// TIA Portal V19 export
FUNCTION "SUGAR" : Void   // FC21, LAD
{ S7_Optimized_Access := 'TRUE' }
// stored: SetENOAutomatically false
   VAR_TEMP   // added for the SCL form of the ladder/FBD networks
      _w1 : Bool;
   END_VAR
BEGIN

REGION Network 1: START MFG PROCESS //////////////////////////////
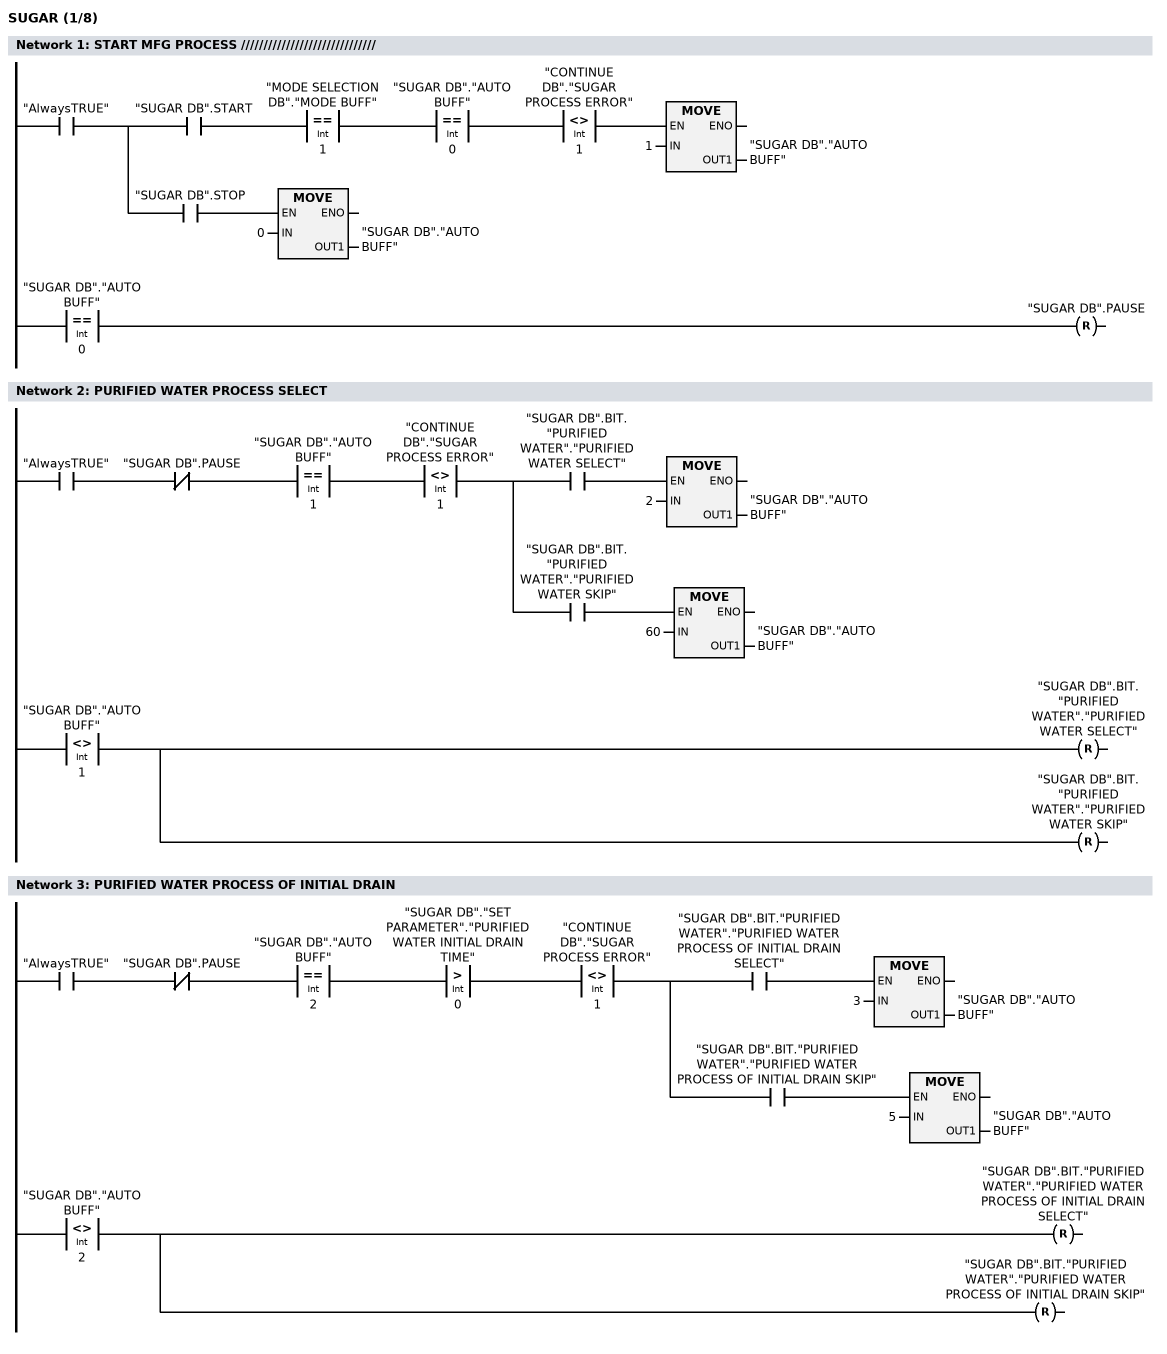
   RUNG wire#powerrail
      Contact( "AlwaysTRUE" )
      wire#w1
      Contact( "SUGAR DB".START )
      { S7_Templates := "SrcType := Int" } EQ_Contact(in1 := "MODE SELECTION DB"."MODE BUFF", in2 := 1)
      { S7_Templates := "SrcType := Int" } EQ_Contact(in1 := "SUGAR DB"."AUTO BUFF", in2 := 0)
      { S7_Templates := "SrcType := Int" } NE_Contact(in1 := "CONTINUE DB"."SUGAR PROCESS ERROR", in2 := 1)
      Move(in := 1, out1 => "SUGAR DB"."AUTO BUFF")
   END_RUNG
   RUNG wire#w1
      Contact( "SUGAR DB".STOP )
      Move(in := 0, out1 => "SUGAR DB"."AUTO BUFF")
   END_RUNG
   RUNG wire#powerrail
      { S7_Templates := "SrcType := Int" } EQ_Contact(in1 := "SUGAR DB"."AUTO BUFF", in2 := 0)
      R_Coil( "SUGAR DB".PAUSE )
   END_RUNG
   // the same network as SCL:
   IF "AlwaysTRUE" AND "SUGAR DB".START AND ("MODE SELECTION DB"."MODE BUFF" = 1) AND ("SUGAR DB"."AUTO BUFF" = 0) AND ("CONTINUE DB"."SUGAR PROCESS ERROR" <> 1) THEN
       "SUGAR DB"."AUTO BUFF" := 1;
   END_IF;
   IF "AlwaysTRUE" AND "SUGAR DB".STOP THEN "SUGAR DB"."AUTO BUFF" := 0; END_IF;
   IF "SUGAR DB"."AUTO BUFF" = 0 THEN "SUGAR DB".PAUSE := FALSE; END_IF;
END_REGION

REGION Network 2: PURIFIED WATER PROCESS SELECT
   RUNG wire#powerrail
      Contact( "AlwaysTRUE" )
      I_Contact( "SUGAR DB".PAUSE )
      { S7_Templates := "SrcType := Int" } EQ_Contact(in1 := "SUGAR DB"."AUTO BUFF", in2 := 1)
      { S7_Templates := "SrcType := Int" } NE_Contact(in1 := "CONTINUE DB"."SUGAR PROCESS ERROR", in2 := 1)
      wire#w1
      Contact( "SUGAR DB".BIT."PURIFIED WATER"."PURIFIED WATER SELECT" )
      Move(in := 2, out1 => "SUGAR DB"."AUTO BUFF")
   END_RUNG
   RUNG wire#w1
      Contact( "SUGAR DB".BIT."PURIFIED WATER"."PURIFIED WATER SKIP" )
      Move(in := 60, out1 => "SUGAR DB"."AUTO BUFF")
   END_RUNG
   RUNG wire#powerrail
      { S7_Templates := "SrcType := Int" } NE_Contact(in1 := "SUGAR DB"."AUTO BUFF", in2 := 1)
      wire#w2
      R_Coil( "SUGAR DB".BIT."PURIFIED WATER"."PURIFIED WATER SELECT" )
   END_RUNG
   RUNG wire#w2
      R_Coil( "SUGAR DB".BIT."PURIFIED WATER"."PURIFIED WATER SKIP" )
   END_RUNG
   // the same network as SCL:
   #_w1 := "AlwaysTRUE" AND NOT "SUGAR DB".PAUSE AND ("SUGAR DB"."AUTO BUFF" = 1) AND ("CONTINUE DB"."SUGAR PROCESS ERROR" <> 1);
   IF #_w1 AND "SUGAR DB".BIT."PURIFIED WATER"."PURIFIED WATER SELECT" THEN
       "SUGAR DB"."AUTO BUFF" := 2;
   END_IF;
   IF #_w1 AND "SUGAR DB".BIT."PURIFIED WATER"."PURIFIED WATER SKIP" THEN
       "SUGAR DB"."AUTO BUFF" := 60;
   END_IF;
   IF "SUGAR DB"."AUTO BUFF" <> 1 THEN
       "SUGAR DB".BIT."PURIFIED WATER"."PURIFIED WATER SELECT" := FALSE;
       "SUGAR DB".BIT."PURIFIED WATER"."PURIFIED WATER SKIP" := FALSE;
   END_IF;
END_REGION

REGION Network 3: PURIFIED WATER PROCESS OF INITIAL DRAIN
   RUNG wire#powerrail
      Contact( "AlwaysTRUE" )
      I_Contact( "SUGAR DB".PAUSE )
      { S7_Templates := "SrcType := Int" } EQ_Contact(in1 := "SUGAR DB"."AUTO BUFF", in2 := 2)
      { S7_Templates := "SrcType := Int" } GT_Contact(in1 := "SUGAR DB"."SET PARAMETER"."PURIFIED WATER INITIAL DRAIN TIME", in2 := 0)
      { S7_Templates := "SrcType := Int" } NE_Contact(in1 := "CONTINUE DB"."SUGAR PROCESS ERROR", in2 := 1)
      wire#w1
      Contact( "SUGAR DB".BIT."PURIFIED WATER"."PURIFIED WATER PROCESS OF INITIAL DRAIN SELECT" )
      Move(in := 3, out1 => "SUGAR DB"."AUTO BUFF")
   END_RUNG
   RUNG wire#w1
      Contact( "SUGAR DB".BIT."PURIFIED WATER"."PURIFIED WATER PROCESS OF INITIAL DRAIN SKIP" )
      Move(in := 5, out1 => "SUGAR DB"."AUTO BUFF")
   END_RUNG
   RUNG wire#powerrail
      { S7_Templates := "SrcType := Int" } NE_Contact(in1 := "SUGAR DB"."AUTO BUFF", in2 := 2)
      wire#w2
      R_Coil( "SUGAR DB".BIT."PURIFIED WATER"."PURIFIED WATER PROCESS OF INITIAL DRAIN SELECT" )
   END_RUNG
   RUNG wire#w2
      R_Coil( "SUGAR DB".BIT."PURIFIED WATER"."PURIFIED WATER PROCESS OF INITIAL DRAIN SKIP" )
   END_RUNG
   // the same network as SCL:
   #_w1 := "AlwaysTRUE" AND NOT "SUGAR DB".PAUSE AND ("SUGAR DB"."AUTO BUFF" = 2) AND ("SUGAR DB"."SET PARAMETER"."PURIFIED WATER INITIAL DRAIN TIME" > 0) AND ("CONTINUE DB"."SUGAR PROCESS ERROR" <> 1);
   IF #_w1 AND "SUGAR DB".BIT."PURIFIED WATER"."PURIFIED WATER PROCESS OF INITIAL DRAIN SELECT" THEN
       "SUGAR DB"."AUTO BUFF" := 3;
   END_IF;
   IF #_w1 AND "SUGAR DB".BIT."PURIFIED WATER"."PURIFIED WATER PROCESS OF INITIAL DRAIN SKIP" THEN
       "SUGAR DB"."AUTO BUFF" := 5;
   END_IF;
   IF "SUGAR DB"."AUTO BUFF" <> 2 THEN
       "SUGAR DB".BIT."PURIFIED WATER"."PURIFIED WATER PROCESS OF INITIAL DRAIN SELECT" := FALSE;
       "SUGAR DB".BIT."PURIFIED WATER"."PURIFIED WATER PROCESS OF INITIAL DRAIN SKIP" := FALSE;
   END_IF;
END_REGION

REGION Network 4: TIMER
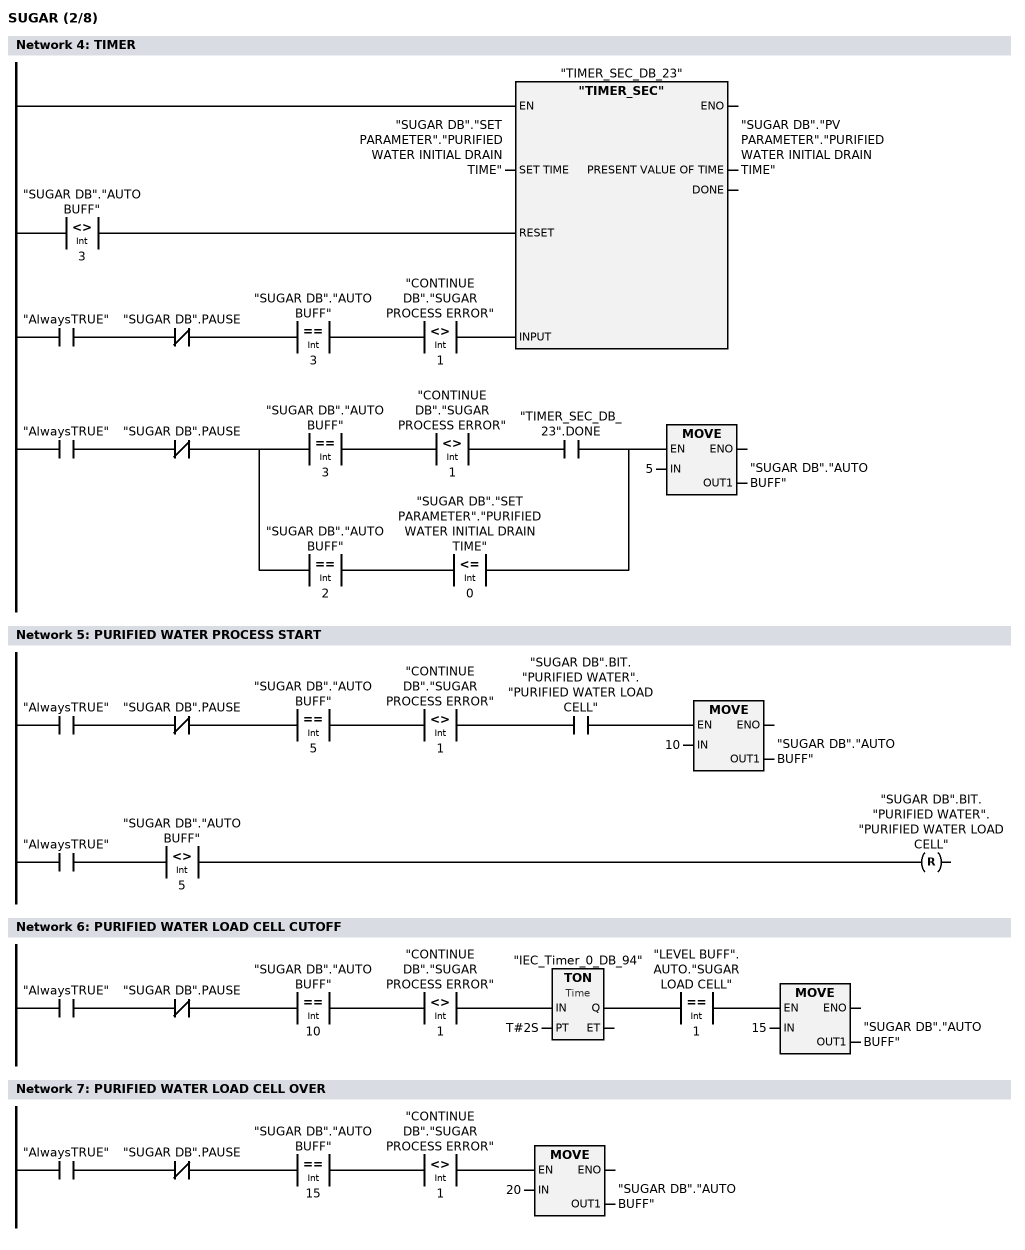
   RUNG wire#powerrail
      "TIMER_SEC_DB_23"(RESET := wire#w1, INPUT := wire#w2, "SET TIME" := "SUGAR DB"."SET PARAMETER"."PURIFIED WATER INITIAL DRAIN TIME", "PRESENT VALUE OF TIME" => "SUGAR DB"."PV PARAMETER"."PURIFIED WATER INITIAL DRAIN TIME", DONE =>)
   END_RUNG
   RUNG wire#powerrail
      { S7_Templates := "SrcType := Int" } NE_Contact(in1 := "SUGAR DB"."AUTO BUFF", in2 := 3)
   END_RUNG wire#w1
   RUNG wire#powerrail
      Contact( "AlwaysTRUE" )
      I_Contact( "SUGAR DB".PAUSE )
      { S7_Templates := "SrcType := Int" } EQ_Contact(in1 := "SUGAR DB"."AUTO BUFF", in2 := 3)
      { S7_Templates := "SrcType := Int" } NE_Contact(in1 := "CONTINUE DB"."SUGAR PROCESS ERROR", in2 := 1)
   END_RUNG wire#w2
   RUNG wire#powerrail
      Contact( "AlwaysTRUE" )
      I_Contact( "SUGAR DB".PAUSE )
      wire#w3
      { S7_Templates := "SrcType := Int" } EQ_Contact(in1 := "SUGAR DB"."AUTO BUFF", in2 := 3)
      { S7_Templates := "SrcType := Int" } NE_Contact(in1 := "CONTINUE DB"."SUGAR PROCESS ERROR", in2 := 1)
      Contact( "TIMER_SEC_DB_23".DONE )
      wire#w4
      Move(in := 5, out1 => "SUGAR DB"."AUTO BUFF")
   END_RUNG
   RUNG wire#w3
      { S7_Templates := "SrcType := Int" } EQ_Contact(in1 := "SUGAR DB"."AUTO BUFF", in2 := 2)
      { S7_Templates := "SrcType := Int" } LE_Contact(in1 := "SUGAR DB"."SET PARAMETER"."PURIFIED WATER INITIAL DRAIN TIME", in2 := 0)
   END_RUNG wire#w4
   // the same network as SCL:
   "TIMER_SEC_DB_23"("SET TIME" := "SUGAR DB"."SET PARAMETER"."PURIFIED WATER INITIAL DRAIN TIME",   // "TIMER_SEC"
                     RESET := "SUGAR DB"."AUTO BUFF" <> 3,
                     INPUT := "AlwaysTRUE" AND NOT "SUGAR DB".PAUSE AND ("SUGAR DB"."AUTO BUFF" = 3) AND ("CONTINUE DB"."SUGAR PROCESS ERROR" <> 1),
                     "PRESENT VALUE OF TIME" => "SUGAR DB"."PV PARAMETER"."PURIFIED WATER INITIAL DRAIN TIME");
   IF "AlwaysTRUE" AND NOT "SUGAR DB".PAUSE AND ((("SUGAR DB"."AUTO BUFF" = 3) AND ("CONTINUE DB"."SUGAR PROCESS ERROR" <> 1) AND "TIMER_SEC_DB_23".DONE) OR (("SUGAR DB"."AUTO BUFF" = 2) AND ("SUGAR DB"."SET PARAMETER"."PURIFIED WATER INITIAL DRAIN TIME" <= 0))) THEN
       "SUGAR DB"."AUTO BUFF" := 5;
   END_IF;
END_REGION

REGION Network 5: PURIFIED WATER PROCESS START
   RUNG wire#powerrail
      Contact( "AlwaysTRUE" )
      I_Contact( "SUGAR DB".PAUSE )
      { S7_Templates := "SrcType := Int" } EQ_Contact(in1 := "SUGAR DB"."AUTO BUFF", in2 := 5)
      { S7_Templates := "SrcType := Int" } NE_Contact(in1 := "CONTINUE DB"."SUGAR PROCESS ERROR", in2 := 1)
      Contact( "SUGAR DB".BIT."PURIFIED WATER"."PURIFIED WATER LOAD CELL" )
      Move(in := 10, out1 => "SUGAR DB"."AUTO BUFF")
   END_RUNG
   RUNG wire#powerrail
      Contact( "AlwaysTRUE" )
      { S7_Templates := "SrcType := Int" } NE_Contact(in1 := "SUGAR DB"."AUTO BUFF", in2 := 5)
      R_Coil( "SUGAR DB".BIT."PURIFIED WATER"."PURIFIED WATER LOAD CELL" )
   END_RUNG
   // the same network as SCL:
   IF "AlwaysTRUE" AND NOT "SUGAR DB".PAUSE AND ("SUGAR DB"."AUTO BUFF" = 5) AND ("CONTINUE DB"."SUGAR PROCESS ERROR" <> 1) AND "SUGAR DB".BIT."PURIFIED WATER"."PURIFIED WATER LOAD CELL" THEN
       "SUGAR DB"."AUTO BUFF" := 10;
   END_IF;
   IF "AlwaysTRUE" AND ("SUGAR DB"."AUTO BUFF" <> 5) THEN
       "SUGAR DB".BIT."PURIFIED WATER"."PURIFIED WATER LOAD CELL" := FALSE;
   END_IF;
END_REGION

REGION Network 6: PURIFIED WATER LOAD CELL CUTOFF
   RUNG wire#powerrail
      Contact( "AlwaysTRUE" )
      I_Contact( "SUGAR DB".PAUSE )
      { S7_Templates := "SrcType := Int" } EQ_Contact(in1 := "SUGAR DB"."AUTO BUFF", in2 := 10)
      { S7_Templates := "SrcType := Int" } NE_Contact(in1 := "CONTINUE DB"."SUGAR PROCESS ERROR", in2 := 1)
      { S7_Templates := "time_type := Time" } "IEC_Timer_0_DB_94".TON(pt := T#2S, et =>)
      { S7_Templates := "SrcType := Int" } EQ_Contact(in1 := "LEVEL BUFF".AUTO."SUGAR LOAD CELL", in2 := 1)
      Move(in := 15, out1 => "SUGAR DB"."AUTO BUFF")
   END_RUNG
   // the same network as SCL:
   "IEC_Timer_0_DB_94".TON(IN := "AlwaysTRUE" AND NOT "SUGAR DB".PAUSE AND ("SUGAR DB"."AUTO BUFF" = 10) AND ("CONTINUE DB"."SUGAR PROCESS ERROR" <> 1),
                           PT := T#2S);
   IF "IEC_Timer_0_DB_94".Q AND ("LEVEL BUFF".AUTO."SUGAR LOAD CELL" = 1) THEN
       "SUGAR DB"."AUTO BUFF" := 15;
   END_IF;
END_REGION

REGION Network 7: PURIFIED WATER LOAD CELL OVER
   RUNG wire#powerrail
      Contact( "AlwaysTRUE" )
      I_Contact( "SUGAR DB".PAUSE )
      { S7_Templates := "SrcType := Int" } EQ_Contact(in1 := "SUGAR DB"."AUTO BUFF", in2 := 15)
      { S7_Templates := "SrcType := Int" } NE_Contact(in1 := "CONTINUE DB"."SUGAR PROCESS ERROR", in2 := 1)
      Move(in := 20, out1 => "SUGAR DB"."AUTO BUFF")
   END_RUNG
   // the same network as SCL:
   IF "AlwaysTRUE" AND NOT "SUGAR DB".PAUSE AND ("SUGAR DB"."AUTO BUFF" = 15) AND ("CONTINUE DB"."SUGAR PROCESS ERROR" <> 1) THEN
       "SUGAR DB"."AUTO BUFF" := 20;
   END_IF;
END_REGION

REGION Network 8: PURIFIED WATER HEATING OR COOLING SEL
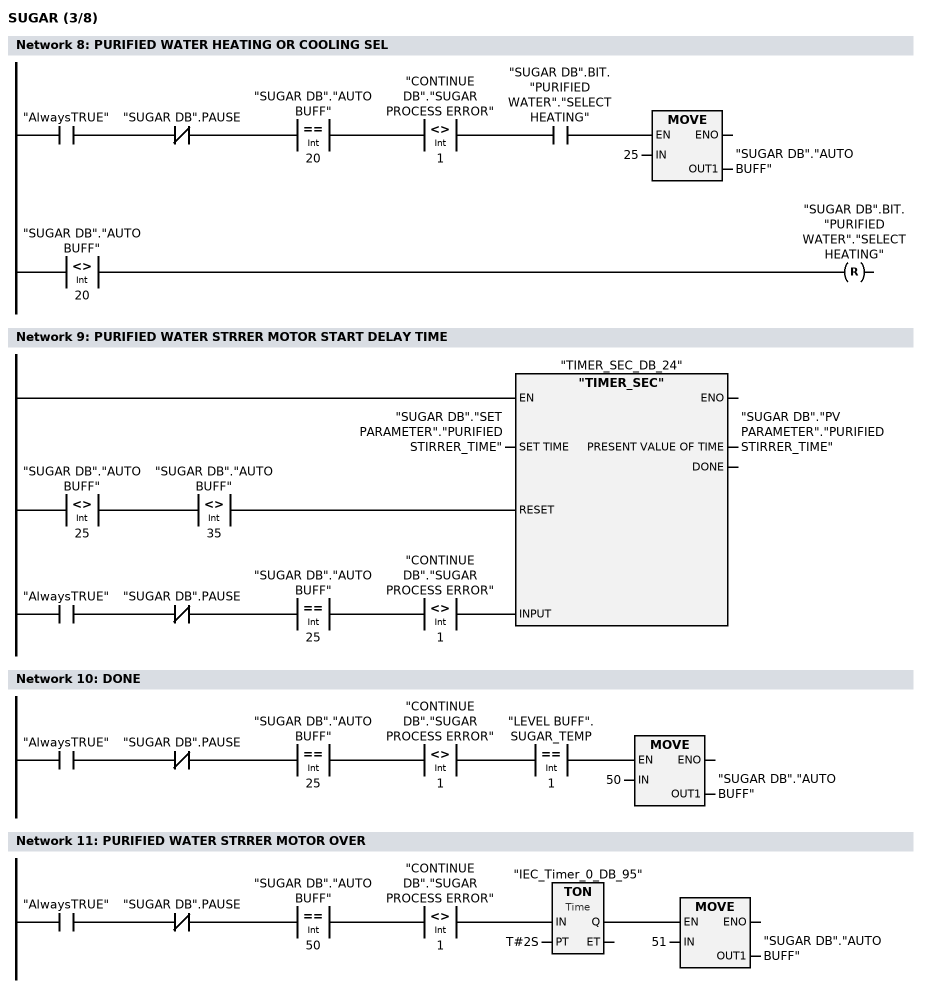
   RUNG wire#powerrail
      Contact( "AlwaysTRUE" )
      I_Contact( "SUGAR DB".PAUSE )
      { S7_Templates := "SrcType := Int" } EQ_Contact(in1 := "SUGAR DB"."AUTO BUFF", in2 := 20)
      { S7_Templates := "SrcType := Int" } NE_Contact(in1 := "CONTINUE DB"."SUGAR PROCESS ERROR", in2 := 1)
      Contact( "SUGAR DB".BIT."PURIFIED WATER"."SELECT HEATING" )
      Move(in := 25, out1 => "SUGAR DB"."AUTO BUFF")
   END_RUNG
   RUNG wire#powerrail
      { S7_Templates := "SrcType := Int" } NE_Contact(in1 := "SUGAR DB"."AUTO BUFF", in2 := 20)
      R_Coil( "SUGAR DB".BIT."PURIFIED WATER"."SELECT HEATING" )
   END_RUNG
   // the same network as SCL:
   IF "AlwaysTRUE" AND NOT "SUGAR DB".PAUSE AND ("SUGAR DB"."AUTO BUFF" = 20) AND ("CONTINUE DB"."SUGAR PROCESS ERROR" <> 1) AND "SUGAR DB".BIT."PURIFIED WATER"."SELECT HEATING" THEN
       "SUGAR DB"."AUTO BUFF" := 25;
   END_IF;
   IF "SUGAR DB"."AUTO BUFF" <> 20 THEN "SUGAR DB".BIT."PURIFIED WATER"."SELECT HEATING" := FALSE; END_IF;
END_REGION

REGION Network 9: PURIFIED WATER STRRER MOTOR START DELAY TIME
   RUNG wire#powerrail
      "TIMER_SEC_DB_24"(RESET := wire#w1, INPUT := wire#w2, "SET TIME" := "SUGAR DB"."SET PARAMETER"."PURIFIED STIRRER_TIME", "PRESENT VALUE OF TIME" => "SUGAR DB"."PV PARAMETER"."PURIFIED STIRRER_TIME", DONE =>)
   END_RUNG
   RUNG wire#powerrail
      { S7_Templates := "SrcType := Int" } NE_Contact(in1 := "SUGAR DB"."AUTO BUFF", in2 := 25)
      { S7_Templates := "SrcType := Int" } NE_Contact(in1 := "SUGAR DB"."AUTO BUFF", in2 := 35)
   END_RUNG wire#w1
   RUNG wire#powerrail
      Contact( "AlwaysTRUE" )
      I_Contact( "SUGAR DB".PAUSE )
      { S7_Templates := "SrcType := Int" } EQ_Contact(in1 := "SUGAR DB"."AUTO BUFF", in2 := 25)
      { S7_Templates := "SrcType := Int" } NE_Contact(in1 := "CONTINUE DB"."SUGAR PROCESS ERROR", in2 := 1)
   END_RUNG wire#w2
   // the same network as SCL:
   "TIMER_SEC_DB_24"("SET TIME" := "SUGAR DB"."SET PARAMETER"."PURIFIED STIRRER_TIME",   // "TIMER_SEC"
                     RESET := ("SUGAR DB"."AUTO BUFF" <> 25) AND ("SUGAR DB"."AUTO BUFF" <> 35),
                     INPUT := "AlwaysTRUE" AND NOT "SUGAR DB".PAUSE AND ("SUGAR DB"."AUTO BUFF" = 25) AND ("CONTINUE DB"."SUGAR PROCESS ERROR" <> 1),
                     "PRESENT VALUE OF TIME" => "SUGAR DB"."PV PARAMETER"."PURIFIED STIRRER_TIME");
END_REGION

REGION Network 10: DONE
   RUNG wire#powerrail
      Contact( "AlwaysTRUE" )
      I_Contact( "SUGAR DB".PAUSE )
      { S7_Templates := "SrcType := Int" } EQ_Contact(in1 := "SUGAR DB"."AUTO BUFF", in2 := 25)
      { S7_Templates := "SrcType := Int" } NE_Contact(in1 := "CONTINUE DB"."SUGAR PROCESS ERROR", in2 := 1)
      { S7_Templates := "SrcType := Int" } EQ_Contact(in1 := "LEVEL BUFF".SUGAR_TEMP, in2 := 1)
      Move(in := 50, out1 => "SUGAR DB"."AUTO BUFF")
   END_RUNG
   // the same network as SCL:
   IF "AlwaysTRUE" AND NOT "SUGAR DB".PAUSE AND ("SUGAR DB"."AUTO BUFF" = 25) AND ("CONTINUE DB"."SUGAR PROCESS ERROR" <> 1) AND ("LEVEL BUFF".SUGAR_TEMP = 1) THEN
       "SUGAR DB"."AUTO BUFF" := 50;
   END_IF;
END_REGION

REGION Network 11: PURIFIED WATER STRRER MOTOR OVER
   RUNG wire#powerrail
      Contact( "AlwaysTRUE" )
      I_Contact( "SUGAR DB".PAUSE )
      { S7_Templates := "SrcType := Int" } EQ_Contact(in1 := "SUGAR DB"."AUTO BUFF", in2 := 50)
      { S7_Templates := "SrcType := Int" } NE_Contact(in1 := "CONTINUE DB"."SUGAR PROCESS ERROR", in2 := 1)
      { S7_Templates := "time_type := Time" } "IEC_Timer_0_DB_95".TON(pt := T#2S, et =>)
      Move(in := 51, out1 => "SUGAR DB"."AUTO BUFF")
   END_RUNG
   // the same network as SCL:
   "IEC_Timer_0_DB_95".TON(IN := "AlwaysTRUE" AND NOT "SUGAR DB".PAUSE AND ("SUGAR DB"."AUTO BUFF" = 50) AND ("CONTINUE DB"."SUGAR PROCESS ERROR" <> 1),
                           PT := T#2S);
   IF "IEC_Timer_0_DB_95".Q THEN "SUGAR DB"."AUTO BUFF" := 51; END_IF;
END_REGION

REGION Network 12: PURIFIED WATER PROCESS OF JACKET DRAIN
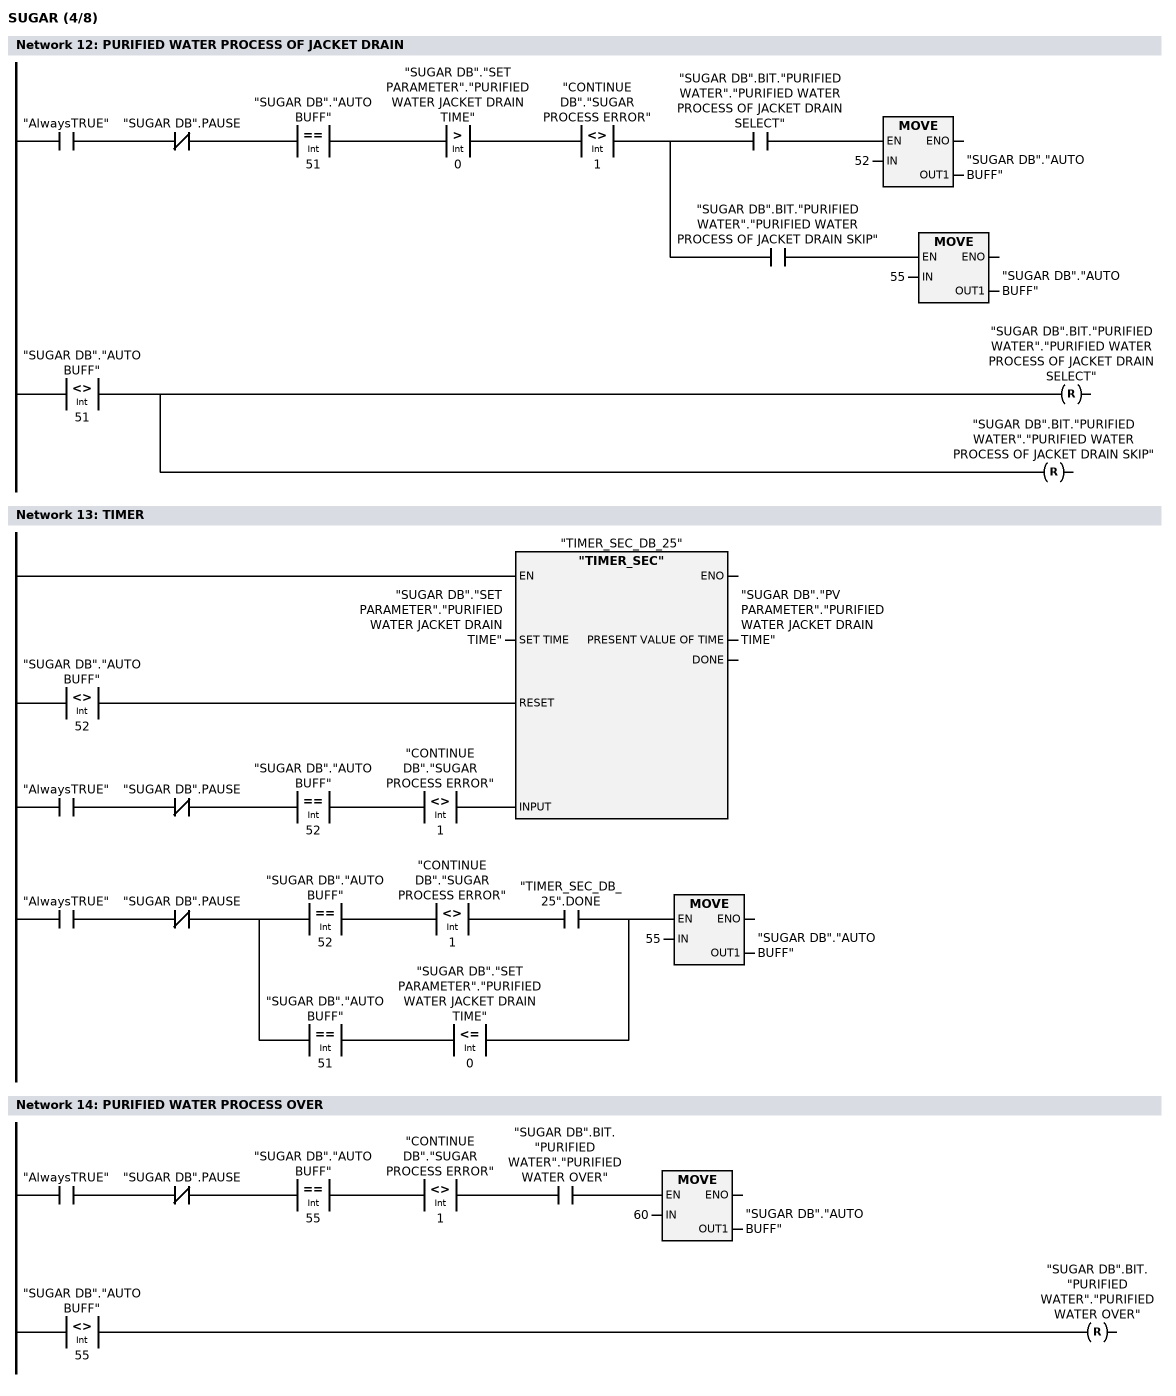
   RUNG wire#powerrail
      Contact( "AlwaysTRUE" )
      I_Contact( "SUGAR DB".PAUSE )
      { S7_Templates := "SrcType := Int" } EQ_Contact(in1 := "SUGAR DB"."AUTO BUFF", in2 := 51)
      { S7_Templates := "SrcType := Int" } GT_Contact(in1 := "SUGAR DB"."SET PARAMETER"."PURIFIED WATER JACKET DRAIN TIME", in2 := 0)
      { S7_Templates := "SrcType := Int" } NE_Contact(in1 := "CONTINUE DB"."SUGAR PROCESS ERROR", in2 := 1)
      wire#w1
      Contact( "SUGAR DB".BIT."PURIFIED WATER"."PURIFIED WATER PROCESS OF JACKET DRAIN SELECT" )
      Move(in := 52, out1 => "SUGAR DB"."AUTO BUFF")
   END_RUNG
   RUNG wire#w1
      Contact( "SUGAR DB".BIT."PURIFIED WATER"."PURIFIED WATER PROCESS OF JACKET DRAIN SKIP" )
      Move(in := 55, out1 => "SUGAR DB"."AUTO BUFF")
   END_RUNG
   RUNG wire#powerrail
      { S7_Templates := "SrcType := Int" } NE_Contact(in1 := "SUGAR DB"."AUTO BUFF", in2 := 51)
      wire#w2
      R_Coil( "SUGAR DB".BIT."PURIFIED WATER"."PURIFIED WATER PROCESS OF JACKET DRAIN SELECT" )
   END_RUNG
   RUNG wire#w2
      R_Coil( "SUGAR DB".BIT."PURIFIED WATER"."PURIFIED WATER PROCESS OF JACKET DRAIN SKIP" )
   END_RUNG
   // the same network as SCL:
   #_w1 := "AlwaysTRUE" AND NOT "SUGAR DB".PAUSE AND ("SUGAR DB"."AUTO BUFF" = 51) AND ("SUGAR DB"."SET PARAMETER"."PURIFIED WATER JACKET DRAIN TIME" > 0) AND ("CONTINUE DB"."SUGAR PROCESS ERROR" <> 1);
   IF #_w1 AND "SUGAR DB".BIT."PURIFIED WATER"."PURIFIED WATER PROCESS OF JACKET DRAIN SELECT" THEN
       "SUGAR DB"."AUTO BUFF" := 52;
   END_IF;
   IF #_w1 AND "SUGAR DB".BIT."PURIFIED WATER"."PURIFIED WATER PROCESS OF JACKET DRAIN SKIP" THEN
       "SUGAR DB"."AUTO BUFF" := 55;
   END_IF;
   IF "SUGAR DB"."AUTO BUFF" <> 51 THEN
       "SUGAR DB".BIT."PURIFIED WATER"."PURIFIED WATER PROCESS OF JACKET DRAIN SELECT" := FALSE;
       "SUGAR DB".BIT."PURIFIED WATER"."PURIFIED WATER PROCESS OF JACKET DRAIN SKIP" := FALSE;
   END_IF;
END_REGION

REGION Network 13: TIMER
   RUNG wire#powerrail
      "TIMER_SEC_DB_25"(RESET := wire#w1, INPUT := wire#w2, "SET TIME" := "SUGAR DB"."SET PARAMETER"."PURIFIED WATER JACKET DRAIN TIME", "PRESENT VALUE OF TIME" => "SUGAR DB"."PV PARAMETER"."PURIFIED WATER JACKET DRAIN TIME", DONE =>)
   END_RUNG
   RUNG wire#powerrail
      { S7_Templates := "SrcType := Int" } NE_Contact(in1 := "SUGAR DB"."AUTO BUFF", in2 := 52)
   END_RUNG wire#w1
   RUNG wire#powerrail
      Contact( "AlwaysTRUE" )
      I_Contact( "SUGAR DB".PAUSE )
      { S7_Templates := "SrcType := Int" } EQ_Contact(in1 := "SUGAR DB"."AUTO BUFF", in2 := 52)
      { S7_Templates := "SrcType := Int" } NE_Contact(in1 := "CONTINUE DB"."SUGAR PROCESS ERROR", in2 := 1)
   END_RUNG wire#w2
   RUNG wire#powerrail
      Contact( "AlwaysTRUE" )
      I_Contact( "SUGAR DB".PAUSE )
      wire#w3
      { S7_Templates := "SrcType := Int" } EQ_Contact(in1 := "SUGAR DB"."AUTO BUFF", in2 := 52)
      { S7_Templates := "SrcType := Int" } NE_Contact(in1 := "CONTINUE DB"."SUGAR PROCESS ERROR", in2 := 1)
      Contact( "TIMER_SEC_DB_25".DONE )
      wire#w4
      Move(in := 55, out1 => "SUGAR DB"."AUTO BUFF")
   END_RUNG
   RUNG wire#w3
      { S7_Templates := "SrcType := Int" } EQ_Contact(in1 := "SUGAR DB"."AUTO BUFF", in2 := 51)
      { S7_Templates := "SrcType := Int" } LE_Contact(in1 := "SUGAR DB"."SET PARAMETER"."PURIFIED WATER JACKET DRAIN TIME", in2 := 0)
   END_RUNG wire#w4
   // the same network as SCL:
   "TIMER_SEC_DB_25"("SET TIME" := "SUGAR DB"."SET PARAMETER"."PURIFIED WATER JACKET DRAIN TIME",   // "TIMER_SEC"
                     RESET := "SUGAR DB"."AUTO BUFF" <> 52,
                     INPUT := "AlwaysTRUE" AND NOT "SUGAR DB".PAUSE AND ("SUGAR DB"."AUTO BUFF" = 52) AND ("CONTINUE DB"."SUGAR PROCESS ERROR" <> 1),
                     "PRESENT VALUE OF TIME" => "SUGAR DB"."PV PARAMETER"."PURIFIED WATER JACKET DRAIN TIME");
   IF "AlwaysTRUE" AND NOT "SUGAR DB".PAUSE AND ((("SUGAR DB"."AUTO BUFF" = 52) AND ("CONTINUE DB"."SUGAR PROCESS ERROR" <> 1) AND "TIMER_SEC_DB_25".DONE) OR (("SUGAR DB"."AUTO BUFF" = 51) AND ("SUGAR DB"."SET PARAMETER"."PURIFIED WATER JACKET DRAIN TIME" <= 0))) THEN
       "SUGAR DB"."AUTO BUFF" := 55;
   END_IF;
END_REGION

REGION Network 14: PURIFIED WATER PROCESS OVER
   RUNG wire#powerrail
      Contact( "AlwaysTRUE" )
      I_Contact( "SUGAR DB".PAUSE )
      { S7_Templates := "SrcType := Int" } EQ_Contact(in1 := "SUGAR DB"."AUTO BUFF", in2 := 55)
      { S7_Templates := "SrcType := Int" } NE_Contact(in1 := "CONTINUE DB"."SUGAR PROCESS ERROR", in2 := 1)
      Contact( "SUGAR DB".BIT."PURIFIED WATER"."PURIFIED WATER OVER" )
      Move(in := 60, out1 => "SUGAR DB"."AUTO BUFF")
   END_RUNG
   RUNG wire#powerrail
      { S7_Templates := "SrcType := Int" } NE_Contact(in1 := "SUGAR DB"."AUTO BUFF", in2 := 55)
      R_Coil( "SUGAR DB".BIT."PURIFIED WATER"."PURIFIED WATER OVER" )
   END_RUNG
   // the same network as SCL:
   IF "AlwaysTRUE" AND NOT "SUGAR DB".PAUSE AND ("SUGAR DB"."AUTO BUFF" = 55) AND ("CONTINUE DB"."SUGAR PROCESS ERROR" <> 1) AND "SUGAR DB".BIT."PURIFIED WATER"."PURIFIED WATER OVER" THEN
       "SUGAR DB"."AUTO BUFF" := 60;
   END_IF;
   IF "SUGAR DB"."AUTO BUFF" <> 55 THEN
       "SUGAR DB".BIT."PURIFIED WATER"."PURIFIED WATER OVER" := FALSE;
   END_IF;
END_REGION

REGION Network 16: MATERIAL SUCTION SELECT / SKIP //////////////////////////////
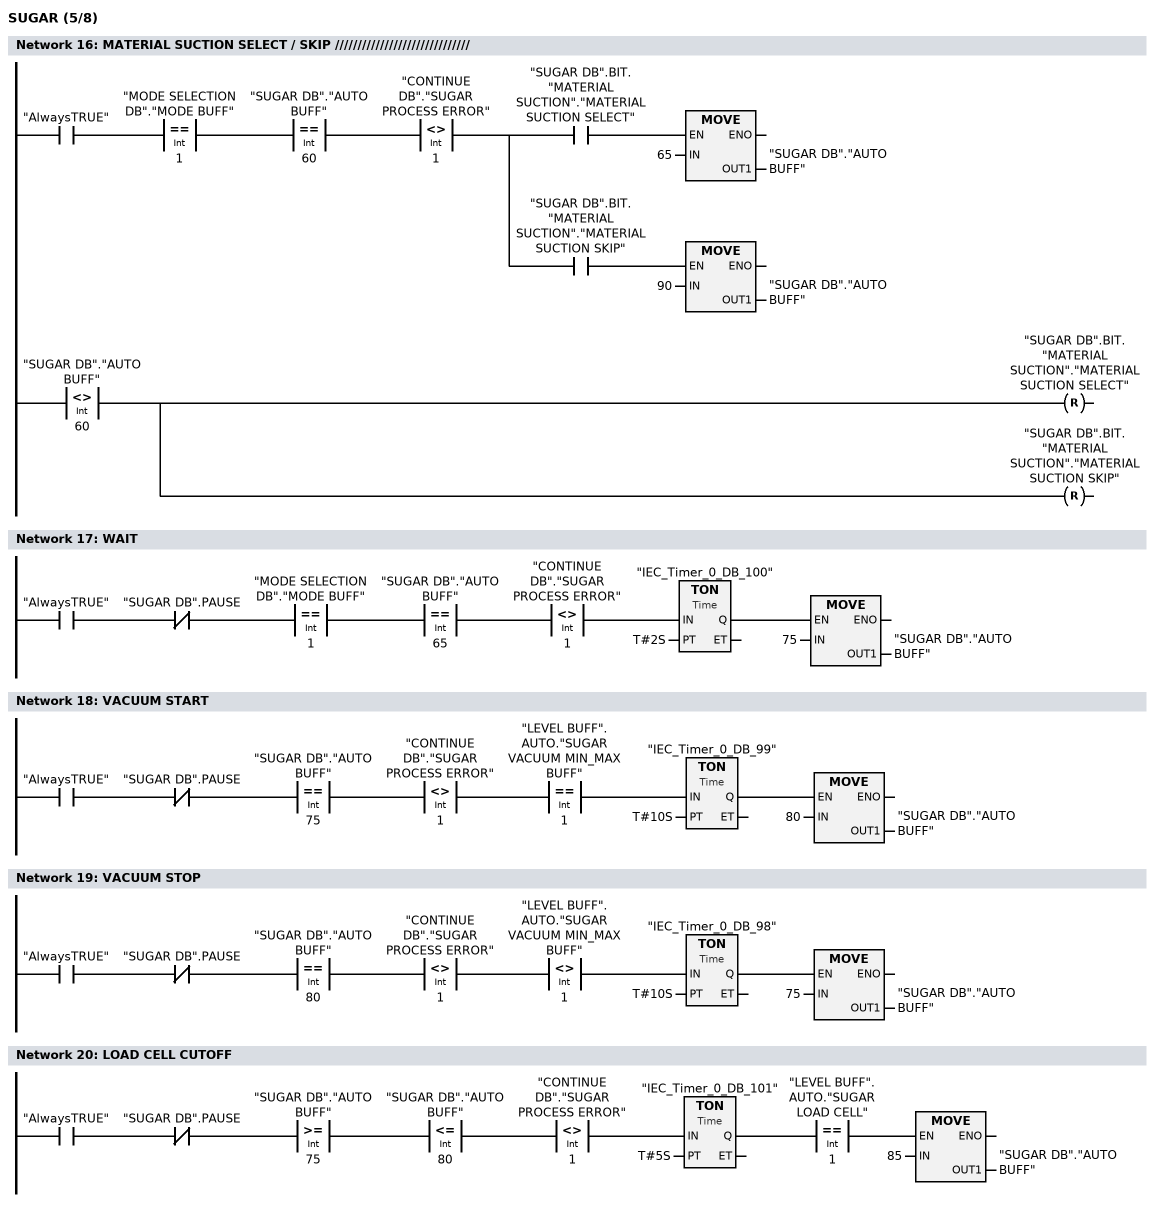
   RUNG wire#powerrail
      Contact( "AlwaysTRUE" )
      { S7_Templates := "SrcType := Int" } EQ_Contact(in1 := "MODE SELECTION DB"."MODE BUFF", in2 := 1)
      { S7_Templates := "SrcType := Int" } EQ_Contact(in1 := "SUGAR DB"."AUTO BUFF", in2 := 60)
      { S7_Templates := "SrcType := Int" } NE_Contact(in1 := "CONTINUE DB"."SUGAR PROCESS ERROR", in2 := 1)
      wire#w1
      Contact( "SUGAR DB".BIT."MATERIAL SUCTION"."MATERIAL SUCTION SELECT" )
      Move(in := 65, out1 => "SUGAR DB"."AUTO BUFF")
   END_RUNG
   RUNG wire#w1
      Contact( "SUGAR DB".BIT."MATERIAL SUCTION"."MATERIAL SUCTION SKIP" )
      Move(in := 90, out1 => "SUGAR DB"."AUTO BUFF")
   END_RUNG
   RUNG wire#powerrail
      { S7_Templates := "SrcType := Int" } NE_Contact(in1 := "SUGAR DB"."AUTO BUFF", in2 := 60)
      wire#w2
      R_Coil( "SUGAR DB".BIT."MATERIAL SUCTION"."MATERIAL SUCTION SELECT" )
   END_RUNG
   RUNG wire#w2
      R_Coil( "SUGAR DB".BIT."MATERIAL SUCTION"."MATERIAL SUCTION SKIP" )
   END_RUNG
   // the same network as SCL:
   #_w1 := "AlwaysTRUE" AND ("MODE SELECTION DB"."MODE BUFF" = 1) AND ("SUGAR DB"."AUTO BUFF" = 60) AND ("CONTINUE DB"."SUGAR PROCESS ERROR" <> 1);
   IF #_w1 AND "SUGAR DB".BIT."MATERIAL SUCTION"."MATERIAL SUCTION SELECT" THEN
       "SUGAR DB"."AUTO BUFF" := 65;
   END_IF;
   IF #_w1 AND "SUGAR DB".BIT."MATERIAL SUCTION"."MATERIAL SUCTION SKIP" THEN
       "SUGAR DB"."AUTO BUFF" := 90;
   END_IF;
   IF "SUGAR DB"."AUTO BUFF" <> 60 THEN
       "SUGAR DB".BIT."MATERIAL SUCTION"."MATERIAL SUCTION SELECT" := FALSE;
       "SUGAR DB".BIT."MATERIAL SUCTION"."MATERIAL SUCTION SKIP" := FALSE;
   END_IF;
END_REGION

REGION Network 17: WAIT
   RUNG wire#powerrail
      Contact( "AlwaysTRUE" )
      I_Contact( "SUGAR DB".PAUSE )
      { S7_Templates := "SrcType := Int" } EQ_Contact(in1 := "MODE SELECTION DB"."MODE BUFF", in2 := 1)
      { S7_Templates := "SrcType := Int" } EQ_Contact(in1 := "SUGAR DB"."AUTO BUFF", in2 := 65)
      { S7_Templates := "SrcType := Int" } NE_Contact(in1 := "CONTINUE DB"."SUGAR PROCESS ERROR", in2 := 1)
      { S7_Templates := "time_type := Time" } "IEC_Timer_0_DB_100".TON(pt := T#2S, et =>)
      Move(in := 75, out1 => "SUGAR DB"."AUTO BUFF")
   END_RUNG
   // the same network as SCL:
   "IEC_Timer_0_DB_100".TON(IN := "AlwaysTRUE" AND NOT "SUGAR DB".PAUSE AND ("MODE SELECTION DB"."MODE BUFF" = 1) AND ("SUGAR DB"."AUTO BUFF" = 65) AND ("CONTINUE DB"."SUGAR PROCESS ERROR" <> 1),
                           PT := T#2S);
   IF "IEC_Timer_0_DB_100".Q THEN "SUGAR DB"."AUTO BUFF" := 75; END_IF;
END_REGION

REGION Network 18: VACUUM START
   RUNG wire#powerrail
      Contact( "AlwaysTRUE" )
      I_Contact( "SUGAR DB".PAUSE )
      { S7_Templates := "SrcType := Int" } EQ_Contact(in1 := "SUGAR DB"."AUTO BUFF", in2 := 75)
      { S7_Templates := "SrcType := Int" } NE_Contact(in1 := "CONTINUE DB"."SUGAR PROCESS ERROR", in2 := 1)
      { S7_Templates := "SrcType := Int" } EQ_Contact(in1 := "LEVEL BUFF".AUTO."SUGAR VACUUM MIN_MAX BUFF", in2 := 1)
      { S7_Templates := "time_type := Time" } "IEC_Timer_0_DB_99".TON(pt := T#10S, et =>)
      Move(in := 80, out1 => "SUGAR DB"."AUTO BUFF")
   END_RUNG
   // the same network as SCL:
   "IEC_Timer_0_DB_99".TON(IN := "AlwaysTRUE" AND NOT "SUGAR DB".PAUSE AND ("SUGAR DB"."AUTO BUFF" = 75) AND ("CONTINUE DB"."SUGAR PROCESS ERROR" <> 1) AND ("LEVEL BUFF".AUTO."SUGAR VACUUM MIN_MAX BUFF" = 1),
                           PT := T#10S);
   IF "IEC_Timer_0_DB_99".Q THEN "SUGAR DB"."AUTO BUFF" := 80; END_IF;
END_REGION

REGION Network 19: VACUUM STOP
   RUNG wire#powerrail
      Contact( "AlwaysTRUE" )
      I_Contact( "SUGAR DB".PAUSE )
      { S7_Templates := "SrcType := Int" } EQ_Contact(in1 := "SUGAR DB"."AUTO BUFF", in2 := 80)
      { S7_Templates := "SrcType := Int" } NE_Contact(in1 := "CONTINUE DB"."SUGAR PROCESS ERROR", in2 := 1)
      { S7_Templates := "SrcType := Int" } NE_Contact(in1 := "LEVEL BUFF".AUTO."SUGAR VACUUM MIN_MAX BUFF", in2 := 1)
      { S7_Templates := "time_type := Time" } "IEC_Timer_0_DB_98".TON(pt := T#10S, et =>)
      Move(in := 75, out1 => "SUGAR DB"."AUTO BUFF")
   END_RUNG
   // the same network as SCL:
   "IEC_Timer_0_DB_98".TON(IN := "AlwaysTRUE" AND NOT "SUGAR DB".PAUSE AND ("SUGAR DB"."AUTO BUFF" = 80) AND ("CONTINUE DB"."SUGAR PROCESS ERROR" <> 1) AND ("LEVEL BUFF".AUTO."SUGAR VACUUM MIN_MAX BUFF" <> 1),
                           PT := T#10S);
   IF "IEC_Timer_0_DB_98".Q THEN "SUGAR DB"."AUTO BUFF" := 75; END_IF;
END_REGION

REGION Network 20: LOAD CELL CUTOFF
   RUNG wire#powerrail
      Contact( "AlwaysTRUE" )
      I_Contact( "SUGAR DB".PAUSE )
      { S7_Templates := "SrcType := Int" } GE_Contact(in1 := "SUGAR DB"."AUTO BUFF", in2 := 75)
      { S7_Templates := "SrcType := Int" } LE_Contact(in1 := "SUGAR DB"."AUTO BUFF", in2 := 80)
      { S7_Templates := "SrcType := Int" } NE_Contact(in1 := "CONTINUE DB"."SUGAR PROCESS ERROR", in2 := 1)
      { S7_Templates := "time_type := Time" } "IEC_Timer_0_DB_101".TON(pt := T#5S, et =>)
      { S7_Templates := "SrcType := Int" } EQ_Contact(in1 := "LEVEL BUFF".AUTO."SUGAR LOAD CELL", in2 := 1)
      Move(in := 85, out1 => "SUGAR DB"."AUTO BUFF")
   END_RUNG
   // the same network as SCL:
   "IEC_Timer_0_DB_101".TON(IN := "AlwaysTRUE" AND NOT "SUGAR DB".PAUSE AND ("SUGAR DB"."AUTO BUFF" >= 75) AND ("SUGAR DB"."AUTO BUFF" <= 80) AND ("CONTINUE DB"."SUGAR PROCESS ERROR" <> 1),
                           PT := T#5S);
   IF "IEC_Timer_0_DB_101".Q AND ("LEVEL BUFF".AUTO."SUGAR LOAD CELL" = 1) THEN
       "SUGAR DB"."AUTO BUFF" := 85;
   END_IF;
END_REGION

REGION Network 21: MATERIAL SUCTION OVER
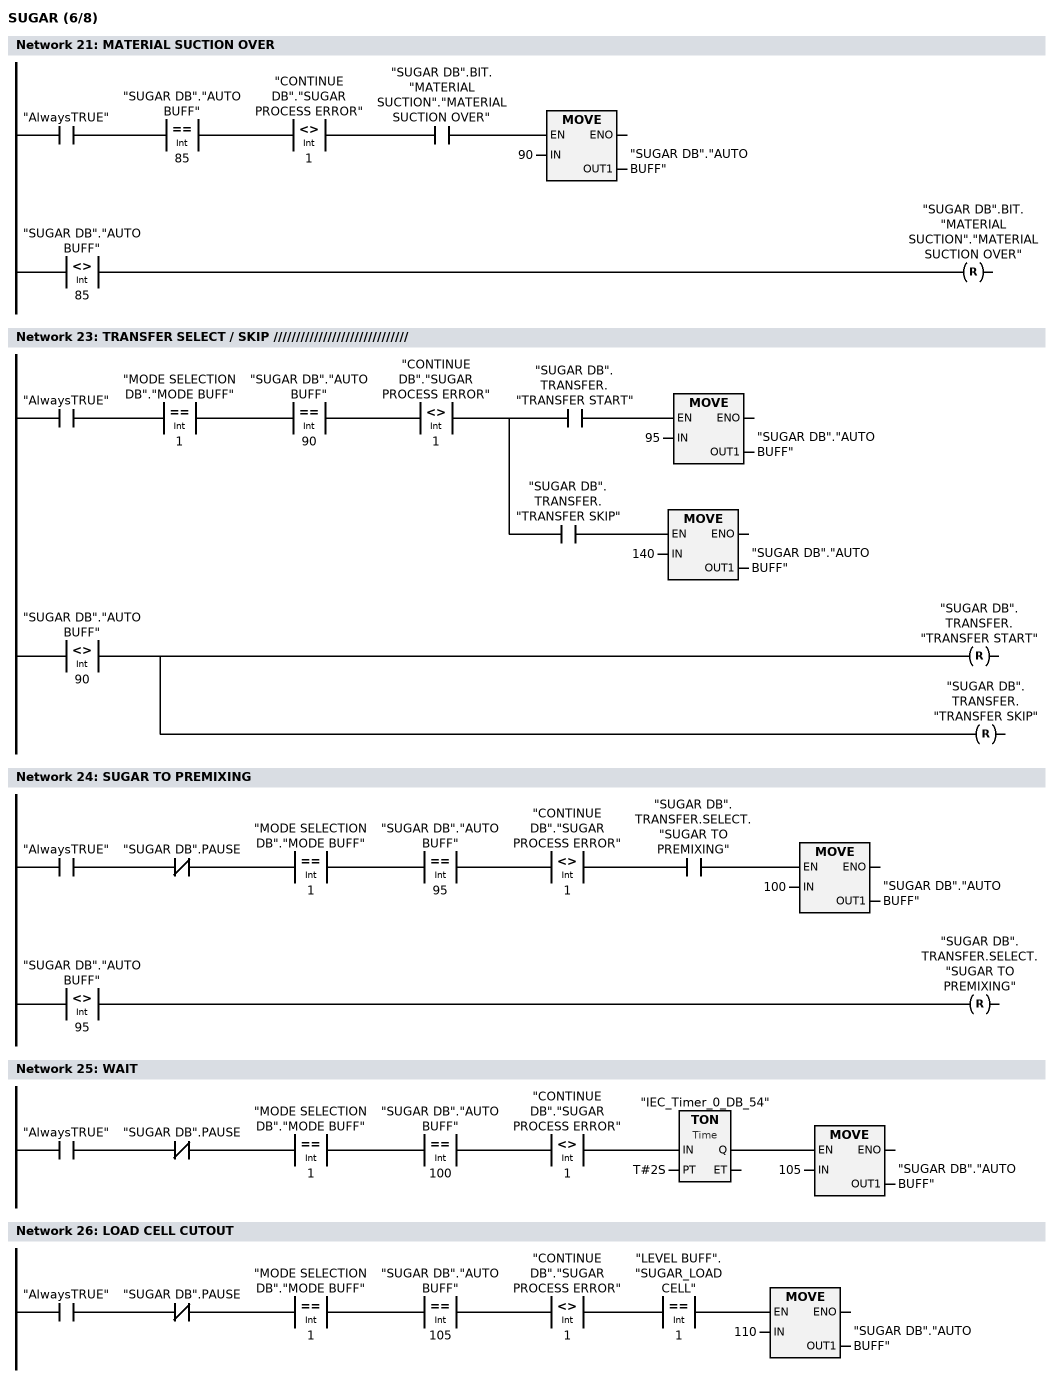
   RUNG wire#powerrail
      Contact( "AlwaysTRUE" )
      { S7_Templates := "SrcType := Int" } EQ_Contact(in1 := "SUGAR DB"."AUTO BUFF", in2 := 85)
      { S7_Templates := "SrcType := Int" } NE_Contact(in1 := "CONTINUE DB"."SUGAR PROCESS ERROR", in2 := 1)
      Contact( "SUGAR DB".BIT."MATERIAL SUCTION"."MATERIAL SUCTION OVER" )
      Move(in := 90, out1 => "SUGAR DB"."AUTO BUFF")
   END_RUNG
   RUNG wire#powerrail
      { S7_Templates := "SrcType := Int" } NE_Contact(in1 := "SUGAR DB"."AUTO BUFF", in2 := 85)
      R_Coil( "SUGAR DB".BIT."MATERIAL SUCTION"."MATERIAL SUCTION OVER" )
   END_RUNG
   // the same network as SCL:
   IF "AlwaysTRUE" AND ("SUGAR DB"."AUTO BUFF" = 85) AND ("CONTINUE DB"."SUGAR PROCESS ERROR" <> 1) AND "SUGAR DB".BIT."MATERIAL SUCTION"."MATERIAL SUCTION OVER" THEN
       "SUGAR DB"."AUTO BUFF" := 90;
   END_IF;
   IF "SUGAR DB"."AUTO BUFF" <> 85 THEN
       "SUGAR DB".BIT."MATERIAL SUCTION"."MATERIAL SUCTION OVER" := FALSE;
   END_IF;
END_REGION

REGION Network 23: TRANSFER SELECT / SKIP //////////////////////////////
   RUNG wire#powerrail
      Contact( "AlwaysTRUE" )
      { S7_Templates := "SrcType := Int" } EQ_Contact(in1 := "MODE SELECTION DB"."MODE BUFF", in2 := 1)
      { S7_Templates := "SrcType := Int" } EQ_Contact(in1 := "SUGAR DB"."AUTO BUFF", in2 := 90)
      { S7_Templates := "SrcType := Int" } NE_Contact(in1 := "CONTINUE DB"."SUGAR PROCESS ERROR", in2 := 1)
      wire#w1
      Contact( "SUGAR DB".TRANSFER."TRANSFER START" )
      Move(in := 95, out1 => "SUGAR DB"."AUTO BUFF")
   END_RUNG
   RUNG wire#w1
      Contact( "SUGAR DB".TRANSFER."TRANSFER SKIP" )
      Move(in := 140, out1 => "SUGAR DB"."AUTO BUFF")
   END_RUNG
   RUNG wire#powerrail
      { S7_Templates := "SrcType := Int" } NE_Contact(in1 := "SUGAR DB"."AUTO BUFF", in2 := 90)
      wire#w2
      R_Coil( "SUGAR DB".TRANSFER."TRANSFER START" )
   END_RUNG
   RUNG wire#w2
      R_Coil( "SUGAR DB".TRANSFER."TRANSFER SKIP" )
   END_RUNG
   // the same network as SCL:
   #_w1 := "AlwaysTRUE" AND ("MODE SELECTION DB"."MODE BUFF" = 1) AND ("SUGAR DB"."AUTO BUFF" = 90) AND ("CONTINUE DB"."SUGAR PROCESS ERROR" <> 1);
   IF #_w1 AND "SUGAR DB".TRANSFER."TRANSFER START" THEN "SUGAR DB"."AUTO BUFF" := 95; END_IF;
   IF #_w1 AND "SUGAR DB".TRANSFER."TRANSFER SKIP" THEN "SUGAR DB"."AUTO BUFF" := 140; END_IF;
   IF "SUGAR DB"."AUTO BUFF" <> 90 THEN
       "SUGAR DB".TRANSFER."TRANSFER START" := FALSE;
       "SUGAR DB".TRANSFER."TRANSFER SKIP" := FALSE;
   END_IF;
END_REGION

REGION Network 24: SUGAR TO PREMIXING
   RUNG wire#powerrail
      Contact( "AlwaysTRUE" )
      I_Contact( "SUGAR DB".PAUSE )
      { S7_Templates := "SrcType := Int" } EQ_Contact(in1 := "MODE SELECTION DB"."MODE BUFF", in2 := 1)
      { S7_Templates := "SrcType := Int" } EQ_Contact(in1 := "SUGAR DB"."AUTO BUFF", in2 := 95)
      { S7_Templates := "SrcType := Int" } NE_Contact(in1 := "CONTINUE DB"."SUGAR PROCESS ERROR", in2 := 1)
      Contact( "SUGAR DB".TRANSFER.SELECT."SUGAR TO PREMIXING" )
      Move(in := 100, out1 => "SUGAR DB"."AUTO BUFF")
   END_RUNG
   RUNG wire#powerrail
      { S7_Templates := "SrcType := Int" } NE_Contact(in1 := "SUGAR DB"."AUTO BUFF", in2 := 95)
      R_Coil( "SUGAR DB".TRANSFER.SELECT."SUGAR TO PREMIXING" )
   END_RUNG
   // the same network as SCL:
   IF "AlwaysTRUE" AND NOT "SUGAR DB".PAUSE AND ("MODE SELECTION DB"."MODE BUFF" = 1) AND ("SUGAR DB"."AUTO BUFF" = 95) AND ("CONTINUE DB"."SUGAR PROCESS ERROR" <> 1) AND "SUGAR DB".TRANSFER.SELECT."SUGAR TO PREMIXING" THEN
       "SUGAR DB"."AUTO BUFF" := 100;
   END_IF;
   IF "SUGAR DB"."AUTO BUFF" <> 95 THEN "SUGAR DB".TRANSFER.SELECT."SUGAR TO PREMIXING" := FALSE; END_IF;
END_REGION

REGION Network 25: WAIT
   RUNG wire#powerrail
      Contact( "AlwaysTRUE" )
      I_Contact( "SUGAR DB".PAUSE )
      { S7_Templates := "SrcType := Int" } EQ_Contact(in1 := "MODE SELECTION DB"."MODE BUFF", in2 := 1)
      { S7_Templates := "SrcType := Int" } EQ_Contact(in1 := "SUGAR DB"."AUTO BUFF", in2 := 100)
      { S7_Templates := "SrcType := Int" } NE_Contact(in1 := "CONTINUE DB"."SUGAR PROCESS ERROR", in2 := 1)
      { S7_Templates := "time_type := Time" } "IEC_Timer_0_DB_54".TON(pt := T#2S, et =>)
      Move(in := 105, out1 => "SUGAR DB"."AUTO BUFF")
   END_RUNG
   // the same network as SCL:
   "IEC_Timer_0_DB_54".TON(IN := "AlwaysTRUE" AND NOT "SUGAR DB".PAUSE AND ("MODE SELECTION DB"."MODE BUFF" = 1) AND ("SUGAR DB"."AUTO BUFF" = 100) AND ("CONTINUE DB"."SUGAR PROCESS ERROR" <> 1),
                           PT := T#2S);
   IF "IEC_Timer_0_DB_54".Q THEN "SUGAR DB"."AUTO BUFF" := 105; END_IF;
END_REGION

REGION Network 26: LOAD CELL CUTOUT
   RUNG wire#powerrail
      Contact( "AlwaysTRUE" )
      I_Contact( "SUGAR DB".PAUSE )
      { S7_Templates := "SrcType := Int" } EQ_Contact(in1 := "MODE SELECTION DB"."MODE BUFF", in2 := 1)
      { S7_Templates := "SrcType := Int" } EQ_Contact(in1 := "SUGAR DB"."AUTO BUFF", in2 := 105)
      { S7_Templates := "SrcType := Int" } NE_Contact(in1 := "CONTINUE DB"."SUGAR PROCESS ERROR", in2 := 1)
      { S7_Templates := "SrcType := Int" } EQ_Contact(in1 := "LEVEL BUFF"."SUGAR_LOAD CELL", in2 := 1)
      Move(in := 110, out1 => "SUGAR DB"."AUTO BUFF")
   END_RUNG
   // the same network as SCL:
   IF "AlwaysTRUE" AND NOT "SUGAR DB".PAUSE AND ("MODE SELECTION DB"."MODE BUFF" = 1) AND ("SUGAR DB"."AUTO BUFF" = 105) AND ("CONTINUE DB"."SUGAR PROCESS ERROR" <> 1) AND ("LEVEL BUFF"."SUGAR_LOAD CELL" = 1) THEN
       "SUGAR DB"."AUTO BUFF" := 110;
   END_IF;
END_REGION

REGION Network 27: TIMER
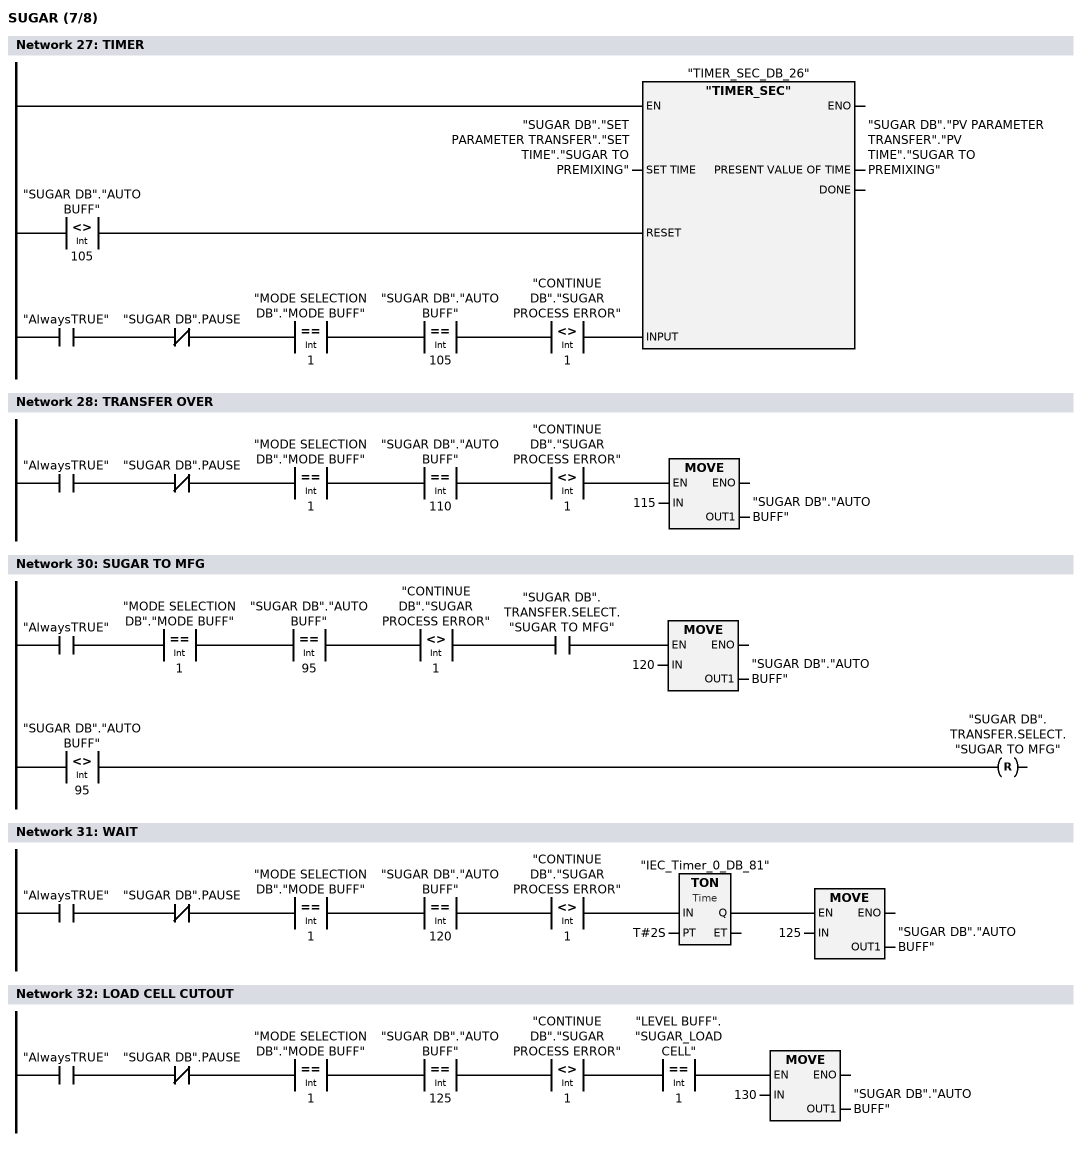
   RUNG wire#powerrail
      "TIMER_SEC_DB_26"(RESET := wire#w1, INPUT := wire#w2, "SET TIME" := "SUGAR DB"."SET PARAMETER TRANSFER"."SET TIME"."SUGAR TO PREMIXING", "PRESENT VALUE OF TIME" => "SUGAR DB"."PV PARAMETER TRANSFER"."PV TIME"."SUGAR TO PREMIXING", DONE =>)
   END_RUNG
   RUNG wire#powerrail
      { S7_Templates := "SrcType := Int" } NE_Contact(in1 := "SUGAR DB"."AUTO BUFF", in2 := 105)
   END_RUNG wire#w1
   RUNG wire#powerrail
      Contact( "AlwaysTRUE" )
      I_Contact( "SUGAR DB".PAUSE )
      { S7_Templates := "SrcType := Int" } EQ_Contact(in1 := "MODE SELECTION DB"."MODE BUFF", in2 := 1)
      { S7_Templates := "SrcType := Int" } EQ_Contact(in1 := "SUGAR DB"."AUTO BUFF", in2 := 105)
      { S7_Templates := "SrcType := Int" } NE_Contact(in1 := "CONTINUE DB"."SUGAR PROCESS ERROR", in2 := 1)
   END_RUNG wire#w2
   // the same network as SCL:
   "TIMER_SEC_DB_26"("SET TIME" := "SUGAR DB"."SET PARAMETER TRANSFER"."SET TIME"."SUGAR TO PREMIXING",   // "TIMER_SEC"
                     RESET := "SUGAR DB"."AUTO BUFF" <> 105,
                     INPUT := "AlwaysTRUE" AND NOT "SUGAR DB".PAUSE AND ("MODE SELECTION DB"."MODE BUFF" = 1) AND ("SUGAR DB"."AUTO BUFF" = 105) AND ("CONTINUE DB"."SUGAR PROCESS ERROR" <> 1),
                     "PRESENT VALUE OF TIME" => "SUGAR DB"."PV PARAMETER TRANSFER"."PV TIME"."SUGAR TO PREMIXING");
END_REGION

REGION Network 28: TRANSFER OVER
   RUNG wire#powerrail
      Contact( "AlwaysTRUE" )
      I_Contact( "SUGAR DB".PAUSE )
      { S7_Templates := "SrcType := Int" } EQ_Contact(in1 := "MODE SELECTION DB"."MODE BUFF", in2 := 1)
      { S7_Templates := "SrcType := Int" } EQ_Contact(in1 := "SUGAR DB"."AUTO BUFF", in2 := 110)
      { S7_Templates := "SrcType := Int" } NE_Contact(in1 := "CONTINUE DB"."SUGAR PROCESS ERROR", in2 := 1)
      Move(in := 115, out1 => "SUGAR DB"."AUTO BUFF")
   END_RUNG
   // the same network as SCL:
   IF "AlwaysTRUE" AND NOT "SUGAR DB".PAUSE AND ("MODE SELECTION DB"."MODE BUFF" = 1) AND ("SUGAR DB"."AUTO BUFF" = 110) AND ("CONTINUE DB"."SUGAR PROCESS ERROR" <> 1) THEN
       "SUGAR DB"."AUTO BUFF" := 115;
   END_IF;
END_REGION

REGION Network 30: SUGAR TO MFG
   RUNG wire#powerrail
      Contact( "AlwaysTRUE" )
      { S7_Templates := "SrcType := Int" } EQ_Contact(in1 := "MODE SELECTION DB"."MODE BUFF", in2 := 1)
      { S7_Templates := "SrcType := Int" } EQ_Contact(in1 := "SUGAR DB"."AUTO BUFF", in2 := 95)
      { S7_Templates := "SrcType := Int" } NE_Contact(in1 := "CONTINUE DB"."SUGAR PROCESS ERROR", in2 := 1)
      Contact( "SUGAR DB".TRANSFER.SELECT."SUGAR TO MFG" )
      Move(in := 120, out1 => "SUGAR DB"."AUTO BUFF")
   END_RUNG
   RUNG wire#powerrail
      { S7_Templates := "SrcType := Int" } NE_Contact(in1 := "SUGAR DB"."AUTO BUFF", in2 := 95)
      R_Coil( "SUGAR DB".TRANSFER.SELECT."SUGAR TO MFG" )
   END_RUNG
   // the same network as SCL:
   IF "AlwaysTRUE" AND ("MODE SELECTION DB"."MODE BUFF" = 1) AND ("SUGAR DB"."AUTO BUFF" = 95) AND ("CONTINUE DB"."SUGAR PROCESS ERROR" <> 1) AND "SUGAR DB".TRANSFER.SELECT."SUGAR TO MFG" THEN
       "SUGAR DB"."AUTO BUFF" := 120;
   END_IF;
   IF "SUGAR DB"."AUTO BUFF" <> 95 THEN "SUGAR DB".TRANSFER.SELECT."SUGAR TO MFG" := FALSE; END_IF;
END_REGION

REGION Network 31: WAIT
   RUNG wire#powerrail
      Contact( "AlwaysTRUE" )
      I_Contact( "SUGAR DB".PAUSE )
      { S7_Templates := "SrcType := Int" } EQ_Contact(in1 := "MODE SELECTION DB"."MODE BUFF", in2 := 1)
      { S7_Templates := "SrcType := Int" } EQ_Contact(in1 := "SUGAR DB"."AUTO BUFF", in2 := 120)
      { S7_Templates := "SrcType := Int" } NE_Contact(in1 := "CONTINUE DB"."SUGAR PROCESS ERROR", in2 := 1)
      { S7_Templates := "time_type := Time" } "IEC_Timer_0_DB_81".TON(pt := T#2S, et =>)
      Move(in := 125, out1 => "SUGAR DB"."AUTO BUFF")
   END_RUNG
   // the same network as SCL:
   "IEC_Timer_0_DB_81".TON(IN := "AlwaysTRUE" AND NOT "SUGAR DB".PAUSE AND ("MODE SELECTION DB"."MODE BUFF" = 1) AND ("SUGAR DB"."AUTO BUFF" = 120) AND ("CONTINUE DB"."SUGAR PROCESS ERROR" <> 1),
                           PT := T#2S);
   IF "IEC_Timer_0_DB_81".Q THEN "SUGAR DB"."AUTO BUFF" := 125; END_IF;
END_REGION

REGION Network 32: LOAD CELL CUTOUT
   RUNG wire#powerrail
      Contact( "AlwaysTRUE" )
      I_Contact( "SUGAR DB".PAUSE )
      { S7_Templates := "SrcType := Int" } EQ_Contact(in1 := "MODE SELECTION DB"."MODE BUFF", in2 := 1)
      { S7_Templates := "SrcType := Int" } EQ_Contact(in1 := "SUGAR DB"."AUTO BUFF", in2 := 125)
      { S7_Templates := "SrcType := Int" } NE_Contact(in1 := "CONTINUE DB"."SUGAR PROCESS ERROR", in2 := 1)
      { S7_Templates := "SrcType := Int" } EQ_Contact(in1 := "LEVEL BUFF"."SUGAR_LOAD CELL", in2 := 1)
      Move(in := 130, out1 => "SUGAR DB"."AUTO BUFF")
   END_RUNG
   // the same network as SCL:
   IF "AlwaysTRUE" AND NOT "SUGAR DB".PAUSE AND ("MODE SELECTION DB"."MODE BUFF" = 1) AND ("SUGAR DB"."AUTO BUFF" = 125) AND ("CONTINUE DB"."SUGAR PROCESS ERROR" <> 1) AND ("LEVEL BUFF"."SUGAR_LOAD CELL" = 1) THEN
       "SUGAR DB"."AUTO BUFF" := 130;
   END_IF;
END_REGION

REGION Network 33: TIMER
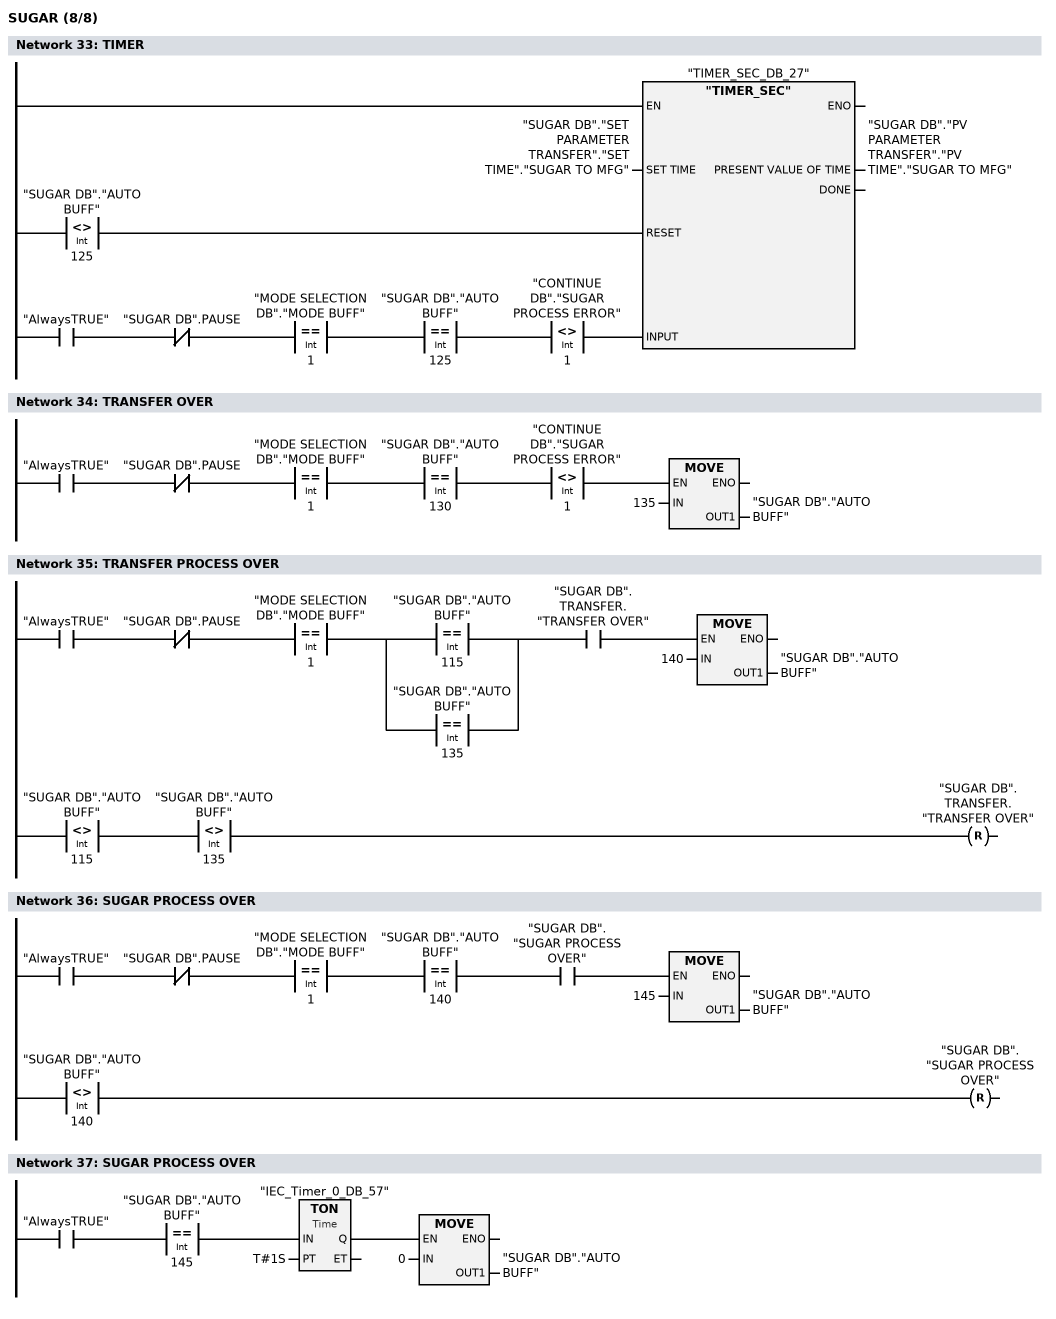
   RUNG wire#powerrail
      "TIMER_SEC_DB_27"(RESET := wire#w1, INPUT := wire#w2, "SET TIME" := "SUGAR DB"."SET PARAMETER TRANSFER"."SET TIME"."SUGAR TO MFG", "PRESENT VALUE OF TIME" => "SUGAR DB"."PV PARAMETER TRANSFER"."PV TIME"."SUGAR TO MFG", DONE =>)
   END_RUNG
   RUNG wire#powerrail
      { S7_Templates := "SrcType := Int" } NE_Contact(in1 := "SUGAR DB"."AUTO BUFF", in2 := 125)
   END_RUNG wire#w1
   RUNG wire#powerrail
      Contact( "AlwaysTRUE" )
      I_Contact( "SUGAR DB".PAUSE )
      { S7_Templates := "SrcType := Int" } EQ_Contact(in1 := "MODE SELECTION DB"."MODE BUFF", in2 := 1)
      { S7_Templates := "SrcType := Int" } EQ_Contact(in1 := "SUGAR DB"."AUTO BUFF", in2 := 125)
      { S7_Templates := "SrcType := Int" } NE_Contact(in1 := "CONTINUE DB"."SUGAR PROCESS ERROR", in2 := 1)
   END_RUNG wire#w2
   // the same network as SCL:
   "TIMER_SEC_DB_27"("SET TIME" := "SUGAR DB"."SET PARAMETER TRANSFER"."SET TIME"."SUGAR TO MFG",   // "TIMER_SEC"
                     RESET := "SUGAR DB"."AUTO BUFF" <> 125,
                     INPUT := "AlwaysTRUE" AND NOT "SUGAR DB".PAUSE AND ("MODE SELECTION DB"."MODE BUFF" = 1) AND ("SUGAR DB"."AUTO BUFF" = 125) AND ("CONTINUE DB"."SUGAR PROCESS ERROR" <> 1),
                     "PRESENT VALUE OF TIME" => "SUGAR DB"."PV PARAMETER TRANSFER"."PV TIME"."SUGAR TO MFG");
END_REGION

REGION Network 34: TRANSFER OVER
   RUNG wire#powerrail
      Contact( "AlwaysTRUE" )
      I_Contact( "SUGAR DB".PAUSE )
      { S7_Templates := "SrcType := Int" } EQ_Contact(in1 := "MODE SELECTION DB"."MODE BUFF", in2 := 1)
      { S7_Templates := "SrcType := Int" } EQ_Contact(in1 := "SUGAR DB"."AUTO BUFF", in2 := 130)
      { S7_Templates := "SrcType := Int" } NE_Contact(in1 := "CONTINUE DB"."SUGAR PROCESS ERROR", in2 := 1)
      Move(in := 135, out1 => "SUGAR DB"."AUTO BUFF")
   END_RUNG
   // the same network as SCL:
   IF "AlwaysTRUE" AND NOT "SUGAR DB".PAUSE AND ("MODE SELECTION DB"."MODE BUFF" = 1) AND ("SUGAR DB"."AUTO BUFF" = 130) AND ("CONTINUE DB"."SUGAR PROCESS ERROR" <> 1) THEN
       "SUGAR DB"."AUTO BUFF" := 135;
   END_IF;
END_REGION

REGION Network 35: TRANSFER PROCESS OVER
   RUNG wire#powerrail
      Contact( "AlwaysTRUE" )
      I_Contact( "SUGAR DB".PAUSE )
      { S7_Templates := "SrcType := Int" } EQ_Contact(in1 := "MODE SELECTION DB"."MODE BUFF", in2 := 1)
      wire#w1
      { S7_Templates := "SrcType := Int" } EQ_Contact(in1 := "SUGAR DB"."AUTO BUFF", in2 := 115)
      wire#w2
      Contact( "SUGAR DB".TRANSFER."TRANSFER OVER" )
      Move(in := 140, out1 => "SUGAR DB"."AUTO BUFF")
   END_RUNG
   RUNG wire#w1
      { S7_Templates := "SrcType := Int" } EQ_Contact(in1 := "SUGAR DB"."AUTO BUFF", in2 := 135)
   END_RUNG wire#w2
   RUNG wire#powerrail
      { S7_Templates := "SrcType := Int" } NE_Contact(in1 := "SUGAR DB"."AUTO BUFF", in2 := 115)
      { S7_Templates := "SrcType := Int" } NE_Contact(in1 := "SUGAR DB"."AUTO BUFF", in2 := 135)
      R_Coil( "SUGAR DB".TRANSFER."TRANSFER OVER" )
   END_RUNG
   // the same network as SCL:
   IF "AlwaysTRUE" AND NOT "SUGAR DB".PAUSE AND ("MODE SELECTION DB"."MODE BUFF" = 1) AND (("SUGAR DB"."AUTO BUFF" = 115) OR ("SUGAR DB"."AUTO BUFF" = 135)) AND "SUGAR DB".TRANSFER."TRANSFER OVER" THEN
       "SUGAR DB"."AUTO BUFF" := 140;
   END_IF;
   IF ("SUGAR DB"."AUTO BUFF" <> 115) AND ("SUGAR DB"."AUTO BUFF" <> 135) THEN
       "SUGAR DB".TRANSFER."TRANSFER OVER" := FALSE;
   END_IF;
END_REGION

REGION Network 36: SUGAR PROCESS OVER
   RUNG wire#powerrail
      Contact( "AlwaysTRUE" )
      I_Contact( "SUGAR DB".PAUSE )
      { S7_Templates := "SrcType := Int" } EQ_Contact(in1 := "MODE SELECTION DB"."MODE BUFF", in2 := 1)
      { S7_Templates := "SrcType := Int" } EQ_Contact(in1 := "SUGAR DB"."AUTO BUFF", in2 := 140)
      Contact( "SUGAR DB"."SUGAR PROCESS OVER" )
      Move(in := 145, out1 => "SUGAR DB"."AUTO BUFF")
   END_RUNG
   RUNG wire#powerrail
      { S7_Templates := "SrcType := Int" } NE_Contact(in1 := "SUGAR DB"."AUTO BUFF", in2 := 140)
      R_Coil( "SUGAR DB"."SUGAR PROCESS OVER" )
   END_RUNG
   // the same network as SCL:
   IF "AlwaysTRUE" AND NOT "SUGAR DB".PAUSE AND ("MODE SELECTION DB"."MODE BUFF" = 1) AND ("SUGAR DB"."AUTO BUFF" = 140) AND "SUGAR DB"."SUGAR PROCESS OVER" THEN
       "SUGAR DB"."AUTO BUFF" := 145;
   END_IF;
   IF "SUGAR DB"."AUTO BUFF" <> 140 THEN "SUGAR DB"."SUGAR PROCESS OVER" := FALSE; END_IF;
END_REGION

REGION Network 37: SUGAR PROCESS OVER
   RUNG wire#powerrail
      Contact( "AlwaysTRUE" )
      { S7_Templates := "SrcType := Int" } EQ_Contact(in1 := "SUGAR DB"."AUTO BUFF", in2 := 145)
      { S7_Templates := "time_type := Time" } "IEC_Timer_0_DB_57".TON(pt := T#1S, et =>)
      Move(in := 0, out1 => "SUGAR DB"."AUTO BUFF")
   END_RUNG
   // the same network as SCL:
   "IEC_Timer_0_DB_57".TON(IN := "AlwaysTRUE" AND ("SUGAR DB"."AUTO BUFF" = 145), PT := T#1S);
   IF "IEC_Timer_0_DB_57".Q THEN "SUGAR DB"."AUTO BUFF" := 0; END_IF;
END_REGION
END_FUNCTION
